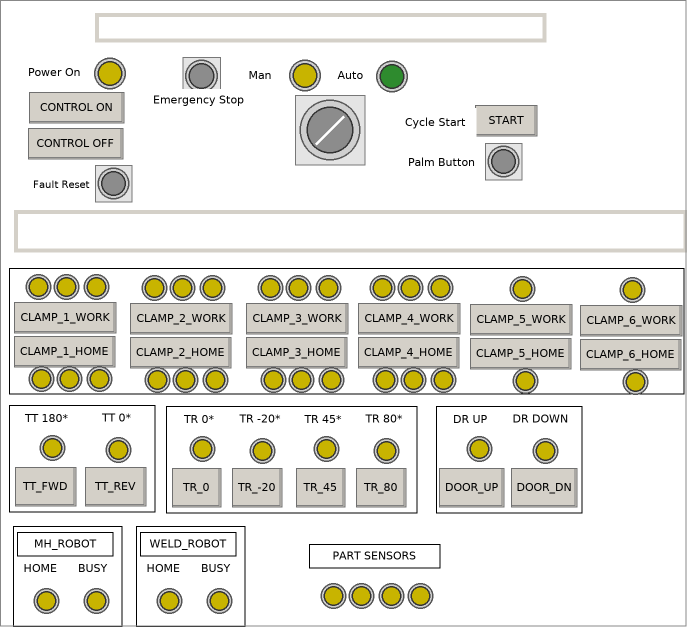
VISUALIZATION Visualization  // 687x627
    Rectangle (13,526 109x101)
    Rectangle (9,405 146x107)
    Rectangle (9,268 675x126)
    Lamp1 (85,55 50x37), variable: Outputs.qPower_On, style: Lamp-Lamp1-Yellow
    Button (29,92 95x31), "CONTROL ON", colour toggle: Inputs.iControl_On, input disabled if: Inputs.iEMR_Stop_PB
        toggle Inputs.iControl_On
    Textfield (24,58 61x29), "Power On"
    Button (28,128 95x31), "CONTROL OFF", colour toggle: Inputs.iControl_OFF
        toggle Inputs.iControl_Off
    RotarySwitch (295,95 70x70), variable: Inputs.iAuto_Manual, behaviour: TOGGLE, style: Switch-RotarySwitch-Gray
    Lamp1 (280,57 50x37), variable: Outputs.qStnMan, style: Lamp-Lamp1-Yellow
    Textfield (244,61 32x29), "Man"
    Lamp1 (367,58 50x37), variable: Outputs.qStnAuto, style: Lamp-Lamp1-Green
    Textfield (334,61 33x29), "Auto"
    Lamp1 (19,272 39x30), variable: Inputs.CC1_Clamp_1_Sensor_WP, style: Lamp-Lamp1-Yellow
    Button (14,302 102x31), "CLAMP_1_WORK", colour toggle: Stn710_DB.CC1_CLAMP.WorkCmd
        tap Stn710_DB.CC1_CLAMP.WorkCmd
    Button (14,336 101x31), "CLAMP_1_HOME", colour toggle: Stn710_DB.CC1_CLAMP.HomeCmd
        tap Stn710_DB.CC1_CLAMP.HomeCmd
    Lamp1 (47,272 39x30), variable: Inputs.CC1_Clamp_2_Sensor_WP, style: Lamp-Lamp1-Yellow
    Lamp1 (77,272 39x30), variable: Inputs.CC1_Clamp_3_Sensor_WP, style: Lamp-Lamp1-Yellow
    Lamp1 (22,364 39x30), variable: Inputs.CC1_Clamp_1_Sensor_HP, style: Lamp-Lamp1-Yellow
    Lamp1 (50,364 39x30), variable: Inputs.CC1_Clamp_2_Sensor_HP, style: Lamp-Lamp1-Yellow
    Lamp1 (80,364 39x30), variable: Inputs.CC1_Clamp_3_Sensor_HP, style: Lamp-Lamp1-Yellow
    PushSwitch (92,165 43x37), variable: Inputs.iResetFault, behaviour: TAP, style: Switch-PushSwitch-Gray
    Textfield (31,170 61x29), "Fault Reset"
    Lamp1 (135,273 39x30), variable: Inputs.CC2_Clamp_1_Sensor_WP, style: Lamp-Lamp1-Yellow
    Button (130,303 102x31), "CLAMP_2_WORK", colour toggle: Stn710_DB.CC2_CLAMP.WorkCmd
        tap Stn710_DB.CC2_CLAMP.WorkCmd
    Button (130,337 101x31), "CLAMP_2_HOME", colour toggle: Stn710_DB.CC2_CLAMP.HomeCmd
        tap Stn710_DB.CC2_CLAMP.HomeCmd
    Lamp1 (163,273 39x30), variable: Inputs.CC2_Clamp_2_Sensor_WP, style: Lamp-Lamp1-Yellow
    Lamp1 (193,273 39x30), variable: Inputs.CC2_Clamp_3_Sensor_WP, style: Lamp-Lamp1-Yellow
    Lamp1 (138,365 39x30), variable: Inputs.CC2_Clamp_1_Sensor_HP, style: Lamp-Lamp1-Yellow
    Lamp1 (166,365 39x30), variable: Inputs.CC2_Clamp_2_Sensor_HP, style: Lamp-Lamp1-Yellow
    Lamp1 (196,365 39x30), variable: Inputs.CC2_Clamp_3_Sensor_HP, style: Lamp-Lamp1-Yellow
    Lamp1 (251,273 39x30), variable: Inputs.CC3_Clamp_1_Sensor_WP, style: Lamp-Lamp1-Yellow
    Button (246,303 102x31), "CLAMP_3_WORK", colour toggle: Stn710_DB.CC3_CLAMP.WorkCmd
        tap Stn710_DB.CC3_CLAMP.WorkCmd
    Button (246,337 101x31), "CLAMP_3_HOME", colour toggle: Stn710_DB.CC3_CLAMP.HomeCmd
        tap Stn710_DB.CC3_CLAMP.HomeCmd
    Lamp1 (279,273 39x30), variable: Inputs.CC3_Clamp_2_Sensor_WP, style: Lamp-Lamp1-Yellow
    Lamp1 (309,273 39x30), variable: Inputs.CC3_Clamp_3_Sensor_WP, style: Lamp-Lamp1-Yellow
    Lamp1 (254,365 39x30), variable: Inputs.CC3_Clamp_1_Sensor_HP, style: Lamp-Lamp1-Yellow
    Lamp1 (282,365 39x30), variable: Inputs.CC3_Clamp_2_Sensor_HP, style: Lamp-Lamp1-Yellow
    Lamp1 (312,365 39x30), variable: Inputs.CC3_Clamp_3_Sensor_HP, style: Lamp-Lamp1-Yellow
    Lamp1 (363,273 39x30), variable: Inputs.CC4_Clamp_1_Sensor_WP, style: Lamp-Lamp1-Yellow
    Button (358,303 102x31), "CLAMP_4_WORK", colour toggle: Stn710_DB.CC4_CLAMP.WorkCmd
        tap Stn710_DB.CC4_CLAMP.WorkCmd
    Button (358,337 101x31), "CLAMP_4_HOME", colour toggle: Stn710_DB.CC4_CLAMP.HomeCmd
        tap Stn710_DB.CC4_CLAMP.HomeCmd
    Lamp1 (391,273 39x30), variable: Inputs.CC4_Clamp_2_Sensor_WP, style: Lamp-Lamp1-Yellow
    Lamp1 (421,273 39x30), variable: Inputs.CC4_Clamp_3_Sensor_WP, style: Lamp-Lamp1-Yellow
    Lamp1 (366,365 39x30), variable: Inputs.CC4_Clamp_1_Sensor_HP, style: Lamp-Lamp1-Yellow
    Lamp1 (394,365 39x30), variable: Inputs.CC4_Clamp_2_Sensor_HP, style: Lamp-Lamp1-Yellow
    Lamp1 (424,365 39x30), variable: Inputs.CC4_Clamp_3_Sensor_HP, style: Lamp-Lamp1-Yellow
    Button (470,304 102x31), "CLAMP_5_WORK", colour toggle: Stn710_DB.CC5_CLAMP.WorkCmd
        tap Stn710_DB.CC5_CLAMP.WorkCmd
    Button (470,338 101x31), "CLAMP_5_HOME", colour toggle: Stn710_DB.CC5_CLAMP.HomeCmd
        tap Stn710_DB.CC5_CLAMP.HomeCmd
    Lamp1 (503,274 39x30), variable: Inputs.CC5_Clamp_1_Sensor_WP, style: Lamp-Lamp1-Yellow
    Lamp1 (506,366 39x30), variable: Inputs.CC5_Clamp_1_Sensor_HP, style: Lamp-Lamp1-Yellow
    Lamp1 (613,275 39x30), variable: Inputs.CC6_Clamp_1_Sensor_WP, style: Lamp-Lamp1-Yellow
    Button (580,305 102x31), "CLAMP_6_WORK", colour toggle: Stn710_DB.CC6_CLAMP.WorkCmd
        tap Stn710_DB.CC6_CLAMP.WorkCmd
    Button (580,339 101x31), "CLAMP_6_HOME", colour toggle: Stn710_DB.CC6_CLAMP.HomeCmd
        tap Stn710_DB.CC6_CLAMP.HomeCmd
    Lamp1 (616,367 39x30), variable: Inputs.CC6_Clamp_1_Sensor_HP, style: Lamp-Lamp1-Yellow
    Button (15,467 61x39), "TT_FWD", colour toggle: Stn710_DB.M_TT_CW
        tap Stn710_DB.M_TT_CW
    Button (85,467 61x39), "TT_REV", colour toggle: Stn710_DB.M_TT_CCW
        tap Stn710_DB.M_TT_CCW
    Lamp1 (33,433 39x30), variable: Stn710_DB.M_TT_FwdSens, style: Lamp-Lamp1-Yellow
    Lamp1 (99,435 39x30), variable: Stn710_DB.M_TT_RevSens, style: Lamp-Lamp1-Yellow
    Textfield (16,409 61x19), "TT 180*"
    Textfield (86,408 61x20), "TT 0*"
    Rectangle (166,406 251x107)
    Button (172,468 49x39), "TR_0", colour toggle: Stn710_DB.M_TR_0_CMD
        tap Stn710_DB.M_TR_0_CMD
    Button (232,468 50x39), "TR_-20", colour toggle: Stn710_DB.M_TR_20_CMD
        tap Stn710_DB.M_TR_20_CMD
    Lamp1 (183,434 39x30), variable: Stn710_DB.M_TR_0_FB, style: Lamp-Lamp1-Yellow
    Lamp1 (243,436 39x30), variable: Stn710_DB.M_TR_20_FB, style: Lamp-Lamp1-Yellow
    Textfield (171,410 56x19), "TR 0*"
    Textfield (235,409 50x20), "TR -20*"
    PushSwitchLed (176,57 51x38), variable: Inputs.iEMR_Stop_PB, behaviour: TOGGLE, style: Switch-PushSwitchLed-Gray
    Textfield (145,89 107x22), "Emergency Stop"
    Rectangle (436,406 146x107)
    Button (439,468 65x39), "DOOR_UP", colour toggle: Stn710_DB.M_DR_UP
        tap Stn710_DB.M_DR_UP
    Button (511,468 66x39), "DOOR_DN", colour toggle: Stn710_DB.M_DR_DOWN
        tap Stn710_DB.M_DR_DOWN
    Lamp1 (460,434 39x30), variable: Stn710_DB.M_DR_UPSens, style: Lamp-Lamp1-Yellow
    Lamp1 (526,436 39x30), variable: Stn710_DB.M_DR_DNSens, style: Lamp-Lamp1-Yellow
    Textfield (443,410 54x19), "DR UP"
    Textfield (507,409 67x20), "DR DOWN"
    Rectangle (17,532 96x24), "MH_ROBOT"
    Textfield (19,559 43x19), "HOME"
    Textfield (73,559 39x19), "BUSY"
    Lamp1 (27,586 39x30), variable: Stn710_DB.MH_RobotHome, style: Lamp-Lamp1-Yellow
    Lamp1 (77,586 39x30), variable: Stn710_DB.MH_RobotBusy, style: Lamp-Lamp1-Yellow
    Rectangle (136,526 109x101)
    Rectangle (140,532 96x24), "WELD_ROBOT"
    Textfield (142,559 43x19), "HOME"
    Textfield (196,559 39x19), "BUSY"
    Lamp1 (150,586 39x30), variable: Stn710_DB.WELD_RobotHome, style: Lamp-Lamp1-Yellow
    Lamp1 (200,586 39x30), variable: Stn710_DB.WELD_RobotBusy, style: Lamp-Lamp1-Yellow
    Textfield (14,210 673x42), text list: 'Seq_list', text index: Auto_Seq_DB.MStep
    Lamp1 (314,581 39x30), variable: Auto_Seq_DB.Part_Sensor1, style: Lamp-Lamp1-Yellow
    Lamp1 (342,581 39x30), variable: Auto_Seq_DB.Part_Sensor2, style: Lamp-Lamp1-Yellow
    Lamp1 (372,581 39x30), variable: Auto_Seq_DB.Part_Sensor3, style: Lamp-Lamp1-Yellow
    Rectangle (309,544 131x24), "PART SENSORS"
    Lamp1 (401,581 39x30), variable: Auto_Seq_DB.Part_Sensor4, style: Lamp-Lamp1-Yellow
    Button (475,105 62x31), "START", colour toggle: Inputs.iCycle_start
        tap Inputs.iCycle_start
    Textfield (401,148 81x29), "Palm Button"
    PushSwitch (482,143 43x37), variable: Inputs.iPalm_Button, behaviour: TAP, style: Switch-PushSwitch-Gray
    Textfield (395,108 81x29), "Cycle Start"
    Textfield (295,410 56x19), "TR 45*"
    Button (296,468 49x39), "TR_45", colour toggle: Stn710_DB.M_TR_45_CMD
        tap Stn710_DB.M_TR_45_CMD
    Button (356,468 50x39), "TR_80", colour toggle: Stn710_DB.M_TR_80_CMD
        tap Stn710_DB.M_TR_80_CMD
    Lamp1 (307,434 39x30), variable: Stn710_DB.M_TR_45_FB, style: Lamp-Lamp1-Yellow
    Lamp1 (367,436 39x30), variable: Stn710_DB.M_TR_80_FB, style: Lamp-Lamp1-Yellow
    Textfield (359,409 50x20), "TR 80*"
    Textfield (95,13 451x29), text list: 'Alarm_list', text index: Stn710_DB.Alarm_count
END_VISUALIZATION

(* stored: Version 1.1.0.1, ProductVersion 3.1.4024.16
   Visu Visualization: Id {b982f27b-3387-4e69-b25f-330d7fd58ebe} *)
